{attribute addProperty BoxType "EK1122-0000-0018"}
{attribute addProperty Id "Beckhoff_ER7xxxsub_EK1100EK1100_179A0949162A_0001_ER7041_0002_0024ER7041_4CF4B42922628.25A_0002_ER7041_0002_0025ER7041_4CF4B42922628.25A_0003_ER7041_1002_0024ER7041_4CF4B42922628.25A_0004_ER7041_1002_0025ER7041_4CF4B42922628.25A_0005_ER7041_2002_0024ER7041_4CF4B42922628.25A_0006_ER7041_2002_0025ER7041_4CF4B42922628.25A_0007_ER7041_3002_0021ER7041_F30AD12822628.25A_0008_ER7041_3002_0022ER7041_F30AD12822628.25A_0009_ER7342_0002_0020ER7342_E03DC37137046.25A_0010_ER7342_0002_0021ER7342_E2585B8337046.25A_0011_ER7342_0002_0022ER7342_E2585B8337046.25"}
{attribute addProperty CRC "3262821403"}
{attribute addProperty SizeInBites "2934"}
{attribute addProperty SizeInBytes "366.75"}
TYPE Beckhoff_ER7xxxEK1122_C27AB41B EXTENDS EK1122_179A0949 :
STRUCT
	{attribute addProperty Name "Beckhoff_ER7xxxsub_EK1100"}
	Beckhoff_ER7xxxsub_EK1100 : EK1100_179A0949;
	{attribute addProperty Name "A_0001_ER7041_0002_0024"}
	A_0001_ER7041_0002_0024 : ER7041_4CF4B429;
	{attribute addProperty Name "A_0002_ER7041_0002_0025"}
	A_0002_ER7041_0002_0025 : ER7041_4CF4B429;
	{attribute addProperty Name "A_0003_ER7041_1002_0024"}
	A_0003_ER7041_1002_0024 : ER7041_4CF4B429;
	{attribute addProperty Name "A_0004_ER7041_1002_0025"}
	A_0004_ER7041_1002_0025 : ER7041_4CF4B429;
	{attribute addProperty Name "A_0005_ER7041_2002_0024"}
	A_0005_ER7041_2002_0024 : ER7041_4CF4B429;
	{attribute addProperty Name "A_0006_ER7041_2002_0025"}
	A_0006_ER7041_2002_0025 : ER7041_4CF4B429;
	{attribute addProperty Name "A_0007_ER7041_3002_0021"}
	A_0007_ER7041_3002_0021 : ER7041_F30AD128;
	{attribute addProperty Name "A_0008_ER7041_3002_0022"}
	A_0008_ER7041_3002_0022 : ER7041_F30AD128;
	{attribute addProperty Name "A_0009_ER7342_0002_0020"}
	A_0009_ER7342_0002_0020 : ER7342_E03DC371;
	{attribute addProperty Name "A_0010_ER7342_0002_0021"}
	A_0010_ER7342_0002_0021 : ER7342_E2585B83;
	{attribute addProperty Name "A_0011_ER7342_0002_0022"}
	A_0011_ER7342_0002_0022 : ER7342_E2585B83;
END_STRUCT
END_TYPE

(* stored: Version 1.2.0.0, ProductVersion 3.1.4024.9
   DUT Beckhoff_ER7xxxEK1122_C27AB41B: Id {78e6b3eb-cf2a-479b-933d-ab41e6219a70} *)
